// TIA Portal V21 export
TYPE "motorStatus"
   STRUCT
      ready : Bool;
      operation : Bool;
      runFwd : Bool;
      runRev : Bool;
      alm : Bool;
      unackAlm : Bool;
   END_STRUCT;
END_TYPE
